FUNCTION_BLOCK FB_Test2
VAR_INPUT
	bTest : INT;
END_VAR
VAR_OUTPUT
	bOut : INT;
END_VAR
VAR
END_VAR

bOut := 2*bTest;

END_FUNCTION_BLOCK

(* stored: Version 1.1.0.1, ProductVersion 3.1.4024.12
   POU FB_Test2: Id {9bb125dd-180d-4b92-9e89-4d1b14905139}, SpecialFunc None *)
